Universal Robots PolyScope program: Project1pick3.urp

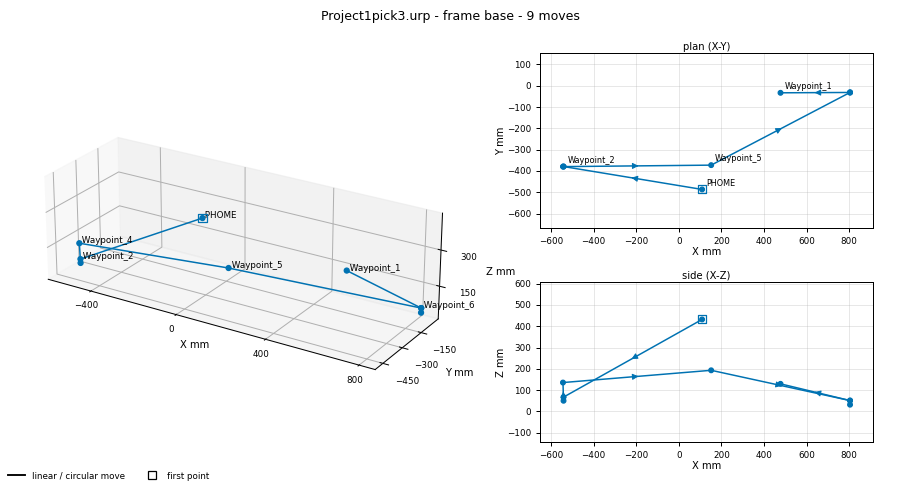
[picture p0: tool path of Project1pick3.urp in frame base, 9 of 9 moves have a stored position in this frame; points joined in program order, loops and branches not executed]
Program Project1pick3 (installation=admin directory=/programs/TUES_530PM createdIn=3.15.8.106339 lastSavedIn=3.15.8.106339 robotSerialNumber=2015350926)
Calibrated DH parameters: a=[0, -0.425, -0.39225, 0, 0, 0]; d=[0.089159, 0, 0, 0.10915, 0.09465, 0.0823]; alpha=[1.570796, 0, 0, 1.570796, -1.570796, 0]; deltaTheta=[0, 0, 0, 0, 0, 0]
Robot Program (runOnlyOnce=true)
  Set DigitalOutput pin=digital_out[0]; digitalValue=0
  MoveL speed 250 mm/s, acceleration 1200 mm/s^2 (useActiveTCP=true) feature=Base
    Waypoint PHOME: TCP in base x=109.128 y=-486.915 z=431.884 mm, rx=0.0001 ry=3.1415 rz=-0.0003 rad; joints [89.997, -90.001, 89.999, -90.008, -89.997, 0] deg
    Waypoint Waypoint_2: TCP in base x=-541.332 y=-379.484 z=67.154 mm, rx=-0.043 ry=3.1175 rz=-0.0122 rad; joints [25.404, -50.501, 93.187, -131.633, -89.023, -66.185] deg
    Waypoint Waypoint_3: TCP in base x=-541.323 y=-379.484 z=50.188 mm, rx=-0.0429 ry=3.1175 rz=-0.0122 rad; joints [25.405, -48.921, 93.501, -133.527, -89.025, -66.18] deg
    Wait Sleep waitTime=0.5
    Set DigitalOutput pin=digital_out[0]; digitalValue=1
    Wait Sleep waitTime=0.5
    Set DigitalOutput pin=digital_out[1]; digitalValue=0
    Wait Sleep waitTime=0.5
    Waypoint Waypoint_4: TCP in base x=-544.016 y=-379.847 z=135.58 mm, rx=-0.0428 ry=3.1081 rz=-0.0056 rad; joints [25.332, -55.975, 90.241, -122.621, -89.022, -66.261] deg
    Waypoint Waypoint_5: TCP in base x=151.728 y=-372.903 z=193.087 mm, rx=-0.0432 ry=3.1279 rz=-0.0102 rad; joints [96.255, -92.567, 130.122, -128.001, -89.27, 4.676] deg
    Waypoint Waypoint_6: TCP in base x=803.616 y=-31.701 z=51.039 mm, rx=2.226 ry=-2.212 rz=0.0054 rad; joints [-190.031, -32.852, 61.234, -118.432, -90.277, -10.391] deg
    Waypoint Waypoint_7: TCP in base x=803.626 y=-31.669 z=31.594 mm, rx=2.2261 ry=-2.2122 rz=0.0055 rad; joints [-190.029, -31.393, 61.498, -120.165, -90.267, -10.388] deg
    Wait Sleep waitTime=0.5
    Set DigitalOutput pin=digital_out[0]; digitalValue=0
    Wait Sleep waitTime=0.5
    Waypoint Waypoint_6: TCP in base x=803.616 y=-31.701 z=51.039 mm, rx=2.226 ry=-2.212 rz=0.0054 rad; joints [-190.031, -32.852, 61.234, -118.432, -90.277, -10.391] deg
    Waypoint Waypoint_1: TCP in base x=477.212 y=-33.349 z=129.551 mm, rx=2.2259 ry=-2.212 rz=0.0053 rad; joints [-197.14, -75.571, 123.035, -137.544, -90.266, -17.499] deg
